(* CODESYS project softmotion.2021.1127.1.project

Project tree, tasks and I/O mapping:
  Device : Changsha-Cyber-MI-linux, Changsha Cyber-MI Co., Ltd., version 3.5.10.40
    application Application
      libraries: Standard, * (System); SysFile, 3.5.15.0 (System); SysTypes2 Interfaces, * (System); SysShm, * (System); CAA Mathematics, * (CAA Technical Workgroup); SysTime, 3.5.9.0 (System); CAA Types Extern, 3.5.13.0 (CAA Technical Workgroup); CAA DTUtil Extern, 3.5.12.0 (CAA Technical Workgroup); Util, * (System); TCP, 3.5.15.0 (3S - Smart Software Solutions GmbH); CAA Net Base Services, 3.5.15.0 (CAA Technical Workgroup); MIC7001 base library, 0.80 (Cyber-MI.com); SM3_CNC_Visu, 4.5.1.0 (3S - Smart Software Solutions GmbH)
      task Task_motion (cyclic, interval 5 ms, priority 9) calls prg_motion, prg_digiout
      task VISU_TASK (cyclic, interval 100 ms, priority 31) calls VisuElems.Visu_Prg
      task Task_prePath (cyclic, interval t#20ms, priority 15) calls prg_prepath
      programs/
        program prg_motion [CFC]
        program prg_prepath [CFC]
      program SoftMotion_PlanningPrg [ST]
      FunctionBlocks/
        function block FB_demo_trafof [ST]
        function block FB_demo_trafo [ST]
      text CNC
      CNC settings
      visualisation Visualization
      trace Trace (task Task_motion): prg_motion.FB_juejinji_trafof_0.x, prg_motion.FB_juejinji_trafof_0.y, prg_motion.FB_juejinji_trafof_0.z
      program prg_digiout [ST]
    SoftMotion General Axis Pool
    IoDrvMIC7001 : IoDrvMIC7001, Cyber-MI, version 19.1.1
        output Application.prg_digiout.do_test : BOOL  // Do03-Ai21@C01
        output Application.prg_digiout.do_test : BOOL  // Do04-Ai22@C03
        output Application.prg_digiout.do_test : BOOL  // Do05-Ai23@C04
        output Application.prg_digiout.do_test : BOOL  // Do06-Ai24@C05
        output Application.prg_digiout.do_test : BOOL  // Do07-Ai25@C06
        output Application.prg_digiout.led_run : BOOL  // LED_run
        unmapped channels: Ai00@C16, Ai01@C28, Ai02@C17, Ai03@C29, Ai04@C30, Ai05@C19, Ai06@C31, Ai07@C20, Ai08@C18, Ai09@D18, Ai10@D20, Ai11@D31, Ai12@D19, Ai13@D30, Ai14@D29, Ai15@D17, Ai16@D28, Ai17@D16, Ai18-Do00@C25, Ai19-Do01@C24, Ai20-Do02@C13, Ai21-Do03@C01, Ai22-Do04@C03, Ai23-Do05@C04, Ai24-Do06@C05, Ai25-Do07@C06, Ai26-Do08@C08, Ai27-Do09@C09, Ai28-Do10@C10, Ai29-Do11@C11, Ai30-Do12@D34, Ai31-Do13@D35, Ai32-Do14@D23, Ai33-Do15@D12, Ai34-Do16@D10, Ai35-Do17@D09, Ai36-Do18@D08, Ai37-Do19@D07, Ai38-Do20@D05, Ai39-Do21@D04,
          Ai40-Do22@D03, Ai41-Do23@D02, Ai42-Do24@C23, Ai43-Do25@C35, Ai44-Do26@D24, Ai45-Do27@D13, Ai46-Ao00@C22, Ai47-Ao01@D14, Ai48_Pi02, Ai49_Out5V, Ai50_VCC, Ai51_VCC_L, Ai52_VCC_R, Ai53_Pwm-i0, Ai54_Pwm-i1, Ai55_Pwm-i2, Ai56_Pwm-i3, Ai57_CPU-T, Ai58_G-x, Ai59_G-y, Ai60_G-z, Ai61-reserved, Ai62-IO-cntr, Ai63-CDS-cntr, Di00-Ai00@C16, Di01-Ai01@C28, Di02-Ai02@C17, Di03-Ai03@C29, Di04-Ai04@C30, Di05-Ai05@C19, Di06-Ai06@C31, Di07-Ai07@C20, Di08-Ai08@C18, Di09-Ai09@D18, Di10-Ai10@D20, Di11-Ai11@D31, Di12-Ai12@D19, Di13-Ai13@D30, Di14-Ai14@D29, Di15-Ai15@D17,
          Di16-Ai16@D28, Di17-Ai17@D16, Di18-Ai18@C25, Di19-Ai19@C24, Di20-Ai20@C13, Di21-Ai21@C01, Di22-Ai22@C03, Di23-Ai23@C04, Di24-Ai24@C05, Di25-Ai25@C06, Di26-Ai26@C08, Di27-Ai27@C09, Di28-Ai28@C10, Di29-Ai29@C11, Di30-Ai30@D34, Di31-Ai31@D35, Di32-Ai32@D23, Di33-Ai33@D12, Di34-Ai34@D10, Di35-Ai35@D09, Di36-Ai36@D08, Di37-Ai37@D07, Di38-Ai38@D05, Di39-Ai39@D04, Di40-Ai40@D03, Di41-Ai41@D02, Di42-Ai42@C23, Di43-Ai43@C35, Di44-Ai44@D24, Di45-Ai45@D13, Di46-Ai46@C22, Di47-Ai47@D14, Di48-Pi00@C15, Di49-Pi01@C14, Di50-Pi02@D22, Di51-Pi03@D21, Di52-reserved, Di53-reserved, Di54-reserved, Di55-reserved,
          Di56-reserved, Di57-reserved, Di58-reserved, Di59-reserved, Di60-reserved, Di61-reserved, Di62-reserved, Di63-reserved, Pi00-Di48@C15, Pi01-Di49@C14, Pi02-Di50@D22, Pi03-Di51@D21, Do00-Ai18@C25, Do01-Ai19@C24, Do02-Ai20@C13, Do08-Ai26@C08, Do09-Ai27@C09, Do10-Ai28@C10, Do11-Ai29@C11, Do12-Ai30@D34, Do13-Ai31@D35, Do14-Ai32@D23, Do15-Ai33@D12, Do16-Ai34@D10, Do17-Ai35@D09, Do18-Ai36@D08, Do19-Ai37@D07, Do20-Ai38@D05, Do21-Ai39@D04, Do22-Ai40@D03, Do23-Ai41@D02, Do24-Ai42@C23, Do25-Ai43@C35, Do26-Ai44@D24, Do27-Ai45@D13, Do28-Pwmi00@C33, Do29-Pwmi01@C34, Do30-Pwmi02@D25, Do31-Pwmi03@D26, PWM00@C25,
          PWM01@C24, PWM02@C13, PWM03@C01, PWM04@C03, PWM05@C04, PWM06@C05, PWM07@C06, PWM08@C08, PWM09@C09, PWM10@C10, PWM11@C11, PWM12@D34, PWM13@D35, PWM14@D23, PWM15@D12, PWM16@D10, PWM17@D09, PWM18@D08, PWM19@D07, PWM20@D05, PWM21@D04, PWM22@D03, PWM23@D02, PWM24@C23, PWM25@C35, PWM26@D24, PWM27@D13, PWM28-Pwmi00@C33, PWM29-Pwmi01@C34, PWM30-Pwmi02@D25, PWM31-Pwmi03@D26, PWM_I_0@C33, PWM_I_1@C34, PWM_I_2@D25, PWM_I_3@D26, Ao00-Ai46@C22, Ao01-Ai47@D14, LED_err, LED_usr, ctrl_ai_raw,
          ctrl_adjust, ctrl_adj0, ctrl_adj1, ctrl_adj2, ctrl_adj3, disable_5V
  libraries: VisuSymbols, 3.5.10.0 (System); SM3_Transformation, 4.5.1.0 (3S - Smart Software Solutions GmbH)
  5ce3da45-db07-42e7-a21c-a00fff4ed8f6|C:\Users\zhou\p01.bmp
  5ce3da45-db07-42e7-a21c-a00fff4ed8f6|C:\working\p01.bmp
  5ce3da45-db07-42e7-a21c-a00fff4ed8f6|C:\working\file.bmp
  text list GlobalTextList
*)

// Device/Application/programs/prg_motion
PROGRAM prg_motion
VAR
	FB_trafo_0: FB_demo_trafo;
	ipo: SMC_Interpolator;
	posinfo:Smc_posinfo;
	
	vc: VisuStruct3DControl;
	
	pt: SMC_PositionTracker;
	pointbuffer_pt: ARRAY [0..1000] OF VisuStruct3DPathPoint;
	
	path_inited :BOOL := FALSE;
	SMC_ReadNCFile_0: SMC_ReadNCFile;
	agcwBufReadNCFile: ARRAY[0..99] OF SMC_GCODE_WORD;
	
	FB_trafof_0: FB_demo_trafof;
END_VAR

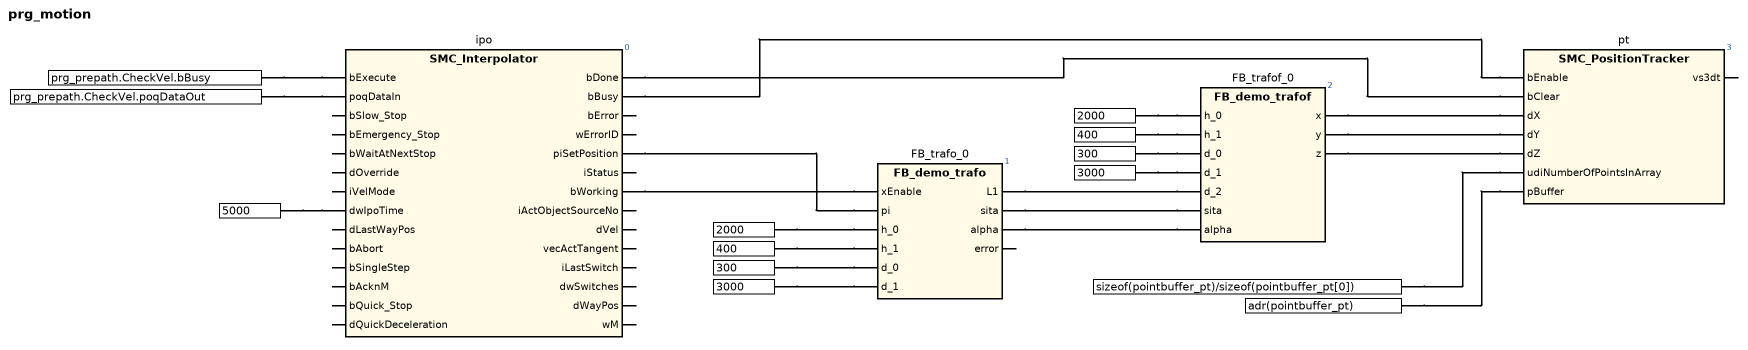
ipo(bExecute := prg_prepath.CheckVel.bBusy, poqDataIn := prg_prepath.CheckVel.poqDataOut, dwIpoTime := 5000); // SMC_Interpolator
FB_trafo_0(
    xEnable := ipo.bWorking,
    pi := ipo.piSetPosition,
    h_0 := 2000,
    h_1 := 400,
    d_0 := 300,
    d_1 := 3000); // FB_demo_trafo
FB_trafof_0(
    h_0 := 2000,
    h_1 := 400,
    d_0 := 300,
    d_1 := 3000,
    d_2 := FB_trafo_0.L1,
    sita := FB_trafo_0.sita,
    alpha := FB_trafo_0.alpha); // FB_demo_trafof
pt(
    bEnable := ipo.bBusy,
    bClear := ipo.bDone,
    dX := FB_trafof_0.x,
    dY := FB_trafof_0.y,
    dZ := FB_trafof_0.z,
    udiNumberOfPointsInArray := sizeof(pointbuffer_pt)/sizeof(pointbuffer_pt[0]),
    pBuffer := adr(pointbuffer_pt)); // SMC_PositionTracker

END_PROGRAM

// Device/Application/programs/prg_prepath
PROGRAM prg_prepath
VAR
	buf1, buf2: ARRAY[0..49] OF SMC_GEOINFO;
	ncDecoder: SMC_NCDecoder;
	SmoothPath: SMC_SmoothPath;
	CheckVel: SMC_CheckVelocities;
	pcf: SMC_PathCopier;
	pointbuffer: ARRAY [0..1000] OF VisuStruct3DPathPoint;
	
	bExe:BOOL := FALSE;
	bApp:BOOL := TRUE;	
	SMC_SmoothPath_0: SMC_SmoothPath;
END_VAR

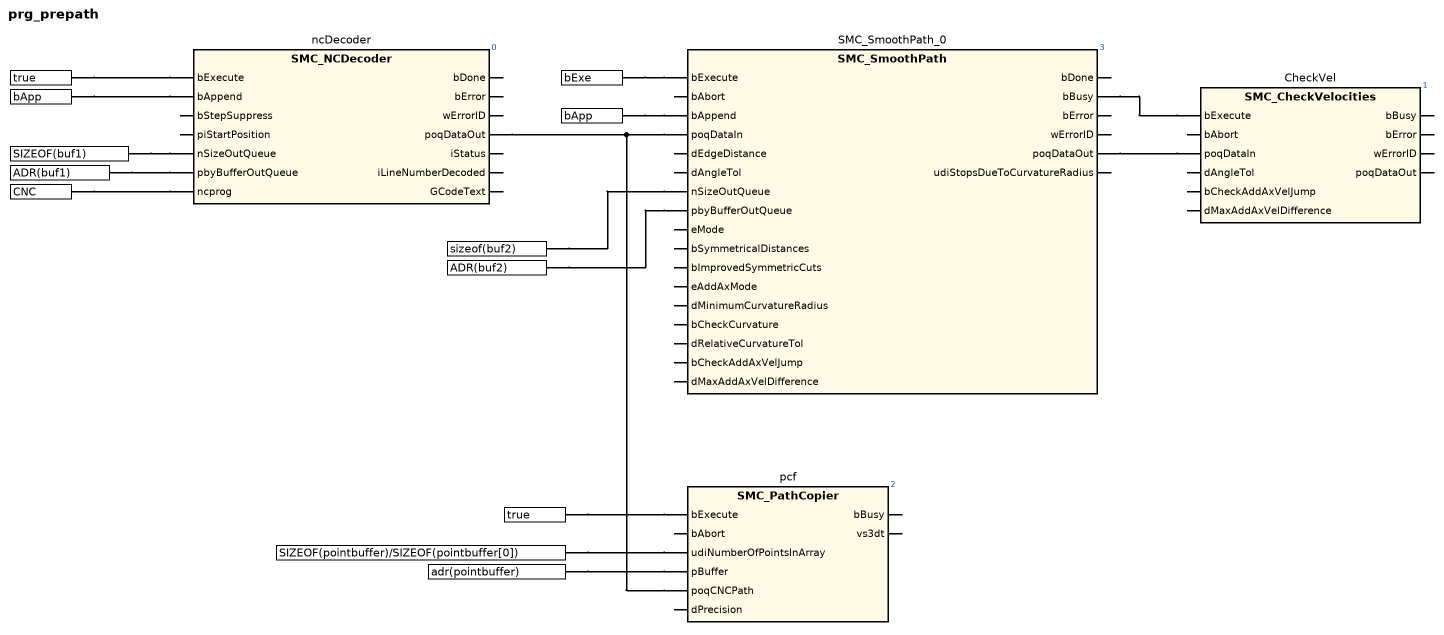
ncDecoder(
    bExecute := true,
    bAppend := bApp,
    nSizeOutQueue := SIZEOF(buf1),
    pbyBufferOutQueue := ADR(buf1),
    ncprog := CNC); // SMC_NCDecoder
CheckVel(bExecute := SMC_SmoothPath_0.bBusy, poqDataIn := SMC_SmoothPath_0.poqDataOut); // SMC_CheckVelocities
pcf(
    bExecute := true,
    udiNumberOfPointsInArray := SIZEOF(pointbuffer)/SIZEOF(pointbuffer[0]),
    pBuffer := adr(pointbuffer),
    poqCNCPath := ncDecoder.poqDataOut); // SMC_PathCopier
SMC_SmoothPath_0(
    bExecute := bExe,
    bAppend := bApp,
    poqDataIn := ncDecoder.poqDataOut,
    nSizeOutQueue := sizeof(buf2),
    pbyBufferOutQueue := ADR(buf2)); // SMC_SmoothPath

END_PROGRAM

// Device/Application/FunctionBlocks/FB_demo_trafo
FUNCTION_BLOCK FB_demo_trafo
VAR_INPUT
	xEnable:BOOL := TRUE;
	pi:SMC_POSINFO;
	h_0:REAL;
	h_1:REAL;
	d_0:REAL;
	d_1:REAL;	
END_VAR
VAR_OUTPUT
	L1:REAL;
	sita:REAL;
	alpha:REAL;
	error:BOOL := FALSE;
END_VAR

VAR
	L : REAL;
	L2 : REAL;
	L3 : REAL;
	
	x:REAL;
	y:REAL;
	z:REAL;
	
	ax:REAL;
	ay:REAL;
	az:REAL;
	
	alpha_0:REAL;  //横臂自身俯仰角
	alpha_1:REAL; //等效俯仰角
	lac:REAL;  //横臂等效长度
	dac:REAL;  //横臂水平长度
	
	xac :REAL;
	yac :REAL;
	zac :REAL;
	
END_VAR

(*  执行机构运动学反变换
 *
 *  点定义：
 *  O:  底座旋转轴在地面的投影点
 *  A： 底座上连接大臂的销轴的中心点
 *  B： 大臂末端截面上的圆心
 *  C： 顶点
 *  
 *  尺寸定义：
 *  h_0: 点 O 到点 A 的垂直距离
 *  h_1: 点 A 到大臂水平状态时中线的垂直距离
 *  d_0: 点 O 到点 A 的水平距离
 *  d_1: 大臂的水平长度， 即点 A 到点 B 的水平距离
 *  d_2: 小臂的实时长度，可伸缩变化
 *
 *  输入： C点的笛卡尔坐标系坐标值（x，y, z)， 基本的机械尺寸
 *  输出： 偏航角： sita，  俯仰角： alpha，  小臂长度： L1
 *  基于三个输出驱动三个油缸进行伺服运动
 *)
IF NOT xEnable THEN
	error := FALSE;
	L1 := 0;
	sita := 0;
	alpha := 0;
	RETURN;
END_IF

x := pi.dX;
y := pi.dY;
z := pi.dZ;

IF ABS(z) < 0.01 THEN
	z := 0.01;
END_IF

sita := ATAN(x/z);  //out 

ax := d_0 * SIN(sita);
ay := h_0;
az := d_0 * COS(sita);

xac := x-ax;
yac := y-ay;
zac := z-az;

alpha_1 := ATAN(yac/zac);
lac := SQRT(xac*xac + yac*yac + zac*zac);
dac := SQRT(lac*lac - h_1*h_1);

L1 := dac - d_1;   //out

alpha_0 := ATAN(h_1/dac);

alpha := alpha_1 - alpha_0;  //out

END_FUNCTION_BLOCK

// Device/Application/FunctionBlocks/FB_demo_trafof
FUNCTION_BLOCK FB_demo_trafof
VAR_INPUT
	h_0:REAL;
	h_1:REAL;
	d_0:REAL;
	d_1:REAL;
	d_2:REAL;
	sita:REAL;  //大臂偏航角度，向前为0度，右转为正
	alpha:REAL;  //大臂俯仰角度，向前为0度，上抬为正
END_VAR
VAR_OUTPUT
	x:REAL;
	y:REAL;
	z:REAL;
END_VAR
VAR
	ax:REAL;
	ay:REAL;
	az:REAL;
	bx:REAL;
	bbY:REAL;
	bz:REAL;
	ab:REAL;
	ac:REAL;
	
	a0:REAL; //大臂自身固有倾角
	a:REAL;  //大臂等效角度
END_VAR

(*  执行机构运动学正变换
 *)
 
ax := d_0 * SIN(sita);
az := d_0 * COS(sita);
ay := h_0;

ab := SQRT(h_1*h_1 + d_1*d_1);

a0 := ATAN(h_1/d_1);
a := a0+alpha;

bx := ax + ab*COS(a)*SIN(sita);
bby:= ay + ab*COS(sita)*SIN(a);
bz := az + ab*COS(a)*COS(sita);

a0 := ATAN(h_1/(d_1+d_2));
a := a0+alpha;

ac := SQRT((d_1+d_2)*(d_1+d_2) + h_1*h_1);

x := ax + ac*COS(a)*SIN(sita);
y := ay + ac*COS(sita)*SIN(a);
z := az + ac*COS(a)*COS(sita);

END_FUNCTION_BLOCK

// Device/Application/prg_digiout
PROGRAM prg_digiout
VAR
	do_test:BOOL:=FALSE;
	led_run:BOOL := TRUE;
	ton_run:ton := (pt := T#500MS);
END_VAR

do_test := TRUE;

ton_run(in := NOT ton_run.Q);
IF ton_run.Q THEN
	led_run := NOT led_run;
END_IF

END_PROGRAM

// Device/Application/SoftMotion_PlanningPrg
PROGRAM SoftMotion_PlanningPrg

;

END_PROGRAM

// Device/Application/Visualization
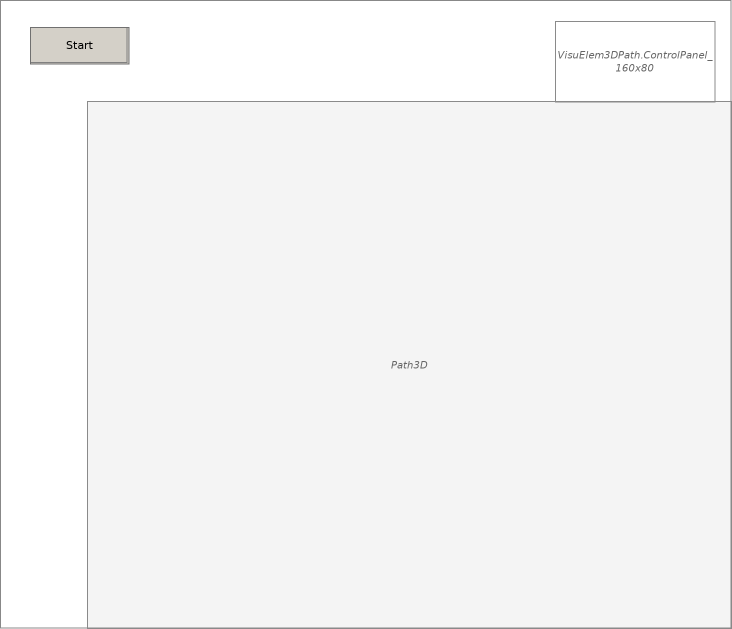
VISUALIZATION Visualization  // 732x629
    Path3D (87,101 645x528)
        p740006429: prg_prepath.pcf.vs3dt
        p81205988: prg_motion.pt.vs3dt
        p3948326086: prg_motion.vc
        p4231319864: prg_motion.ipo.iActObjectSourceNo
    Button (30,27 99x37), "Start"
        toggle prg_prepath.bExe
    Frame (555,21 160x81)
        shows VisuElem3DPath.ControlPanel_160x80(vc := prg_motion.vc)
END_VISUALIZATION

(* text CNC
% 掘进工艺

N00 G92 X0 Y2400 Z4000   					%设定当前坐标，不移动
N10 G01 X-3000 Y500 Z5000 F1250 E30 E-30  	%移动到本次作业的起点： 左下角
N20 G01 X3000  Y500 Z5000   				%第一行作业
N30 G03 Y1000 R250    						%上移到第二行
N40 G01 X-3000        						%第二行作业
N50 G02 Y1500  R250    						%上移到第三行 
N60 G01 X3000          						%第三行作业
N70 G03 Y2000  R250    						%上移到第四行\
N80 G01 X-3000         						%第四行作业
N100 G01 X0 Y2400 Z4000  					%完成本轮作业，回到原点
*)
